DATA_BLOCK "S1.CABINET000.STATE"
{ DB_Accessible_From_OPC_UA := 'FALSE' ;
 S7_Optimized_Access := 'TRUE' }
VERSION : 0.1
NON_RETAIN
"CabState"

BEGIN

END_DATA_BLOCK

